// TIA Portal V16 export
// export: Created 2021-09-08T12:46:13.0649327Z, ExportSetting WithDefaults, DisplayName Totally Integrated Automation Portal, DisplayVersion V16 Update 3, DisplayName TIA Portal Version Control Interface, DisplayVersion V16 Update 2, DisplayName TIA Portal Openness, DisplayVersion V16 Update 3, DisplayName TIA Portal Teamcenter Gateway, DisplayVersion V16, DisplayName STEP 7 Professional, DisplayVersion V16 Update 3, DisplayName STEP 7 Safety, DisplayVersion V16, DisplayName WinCC Advanced, DisplayVersion V16 Update 3
DATA_BLOCK "dtPropDpump"   // DB21
{ S7_Optimized_Access := 'FALSE' }
VERSION : 0.1
// stored: AutoNumber true, DBAccessibleFromOPCUA true, IsOnlyStoredInLoadMemory false, IsWriteProtectedInAS false
   VAR RETAIN
      dp101 : "PropDosing";
      dp501 : "PropDosing";
      dp502 : "PropDosing";
      dp801 : "PropDosing";
      dp802 : "PropDosing";
      dp803 : "PropDosing";
      dp1001 : "PropDosing";
   END_VAR
BEGIN
END_DATA_BLOCK
